TYPE E_ModeMMA :
(
	Init := 0,
	Auto,
	Man
);
END_TYPE

(* stored: Version 1.1.0.1, ProductVersion 3.1.4020.6
   DUT E_ModeMMA: Id {92388d8d-4225-431c-805a-567ffcd4203f} *)
